Staubli VAL3: motionProgress.pgx

public program motionProgress(num x_nMoveId, num x_nMotProg)
begin

  // Do nothing
  // See start() program for more details

end
